(**************************************************************************************
 * 	Application		:	BoxControl Framework
 *	Revision		:	$Revision: 404529 $
 *	Revision date	:	$Date: 2018-04-23 08:21:38 +0200 (Mo., 23 Apr 2018) $
 *	Last changed by	:	$Author: b7bolm $
 *	URL				:	$URL: http://almscdc.swisslog.com/repo/SWPD/Development/BoxControlFramework/20_Release/trunk/01_Software/BCF/BCF/JumpStart/20_Product/10_App/10_Base/10_Lib/10_Conv/00_GVLs/TU_Table.TcGVL $
 *
 *	Purpose			:	Global variables : Conveyor TU Data
 *
 * ------------------------------------------------------------------------------------
 *	Copyright Swisslog [IP AG], Switzerland. All rights reserved.
 * 
 * ------------------------------------------------------------------------------------
 *	
 * 	Revision History: 
 *
 * 	VERSION			DATE			INITIALS			DESCRIPTION
 *	0.1				01.01.2001		swl					Example
 *
 **************************************************************************************)
VAR_GLOBAL PERSISTENT
	TU_DataTable 	: ARRAY[0..Conveyor.NUMBER_OF_TU_DATA] OF ST_TU_Data; // Contains all TU-data
END_VAR

(* stored: Version 1.1.0.1, ProductVersion 3.1.4022.12
   GVL TU_Table: Id {80374262-b492-40fa-b644-a855e863734c} *)
